{attribute addProperty BoxType "EL6002-0000-0017"}
{attribute addProperty Id "CtrlAT %Q*Ctrl_9717E3671621Data_OutAT %Q*ARRAY[0 ..21] OF USINT176220"}
{attribute addProperty CRC "604386845"}
{attribute addProperty SizeInBites "192"}
{attribute addProperty SizeInBytes "24"}
TYPE COM_RxPDO_Map_Outputs_Channel_85BCA431 :
STRUCT
	{attribute addProperty Name "Ctrl"}
	Ctrl AT %Q* : Ctrl_9717E367;
	{attribute addProperty Name "Data_Out"}
	Data_Out AT %Q* : ARRAY[0 ..21] OF USINT;
END_STRUCT
END_TYPE

(* stored: Version 1.2.0.0, ProductVersion 3.1.4024.9
   DUT COM_RxPDO_Map_Outputs_Channel_85BCA431: Id {95760ffe-b8e2-41c8-8aa7-52e0e7783d9a} *)
